TYPE DUT_STS :
STRUCT
	State : INT;
	ManualMode: BOOL;
	AutoMode: BOOL := TRUE;
	InSimulation: BOOL;
	Closed: BOOL;
	Opening: BOOL;
	Open: BOOL;
	Closing: BOOL;
	Interlock: BOOL;
	Alarm: BOOL;
END_STRUCT
END_TYPE

(* stored: Version 1.1.0.1, ProductVersion 3.1.4024.12
   DUT DUT_STS: Id {0d7fb3f1-0e3b-441c-adba-aed480398811} *)
